// TwinCAT 3 PLC project MicroTestStandATM
// ProgramVersion: 3.1.4020.5
// libraries:
//   lcls-twincat-motion, * (SLAC)
//   lcls2-cc-lib, * (SLAC)
//   Tc2_Standard, * (Beckhoff Automation GmbH)
//   Tc2_System, * (Beckhoff Automation GmbH)
//   Tc2_Utilities, * (Beckhoff Automation GmbH)
//   Tc3_Module, * (Beckhoff Automation GmbH)
//   VisuDialogs
//   VisuSymbols,3.5.10.0,System
// project tree:
//   DUTs/ DUT_MotionStage_Extras.TcDUT (not stored)
//   / GlobalTextList.TcGTLO, PlcTask.TcTTO (not stored), VISU_TASK.TcTTO (not stored)
//   POUs/ Main.TcPOU
//   VISUs/ Visualization.TcVIS, VisualizationManager.TcVMO (not stored), VISU_MotionStage.TcVIS (not stored)
// real-time tasks:
//   TASK PlcTask: cycle T#1ms, priority 20, ADS port 350
//   TASK VISU_TASK: cycle T#200000us, priority 30, ADS port 351
// motion (NC):
//   TASK NC-Task 1 SAF: cycle T#1ms, priority 4, ADS port 501
//   TASK NC-Task 1 SVB: cycle T#1ms, priority 8, ADS port 511
//   AXIS MMS_Y (id 1)
//     Dynamic: AccelerationMaximum=200, DecelerationMaximum=200, Acceleration=200, Deceleration=200, Jerk=500, DelayTime=0.004
//     Velo: Maximum=65
//     TargetPosControl: Range=0.002, Time=0.25
//     OtherSettings: AllowMotionCmdToSlave=true
//     encoder EncType=29
//       EncPara: ScaleFactorNumerator=5e-05, Offset=-214686.941, MaxCount=#xffffffff, ReferenceSystem=1
//         Inc: RefSoftSyncMask=#x0000ffff
//     drive DrvType=24
//       Analog: VeloReferenz=100, ScaleFactorActTorque=0.1
//       TimeComp: TaskDelayCycles=1
//     controller CtrType=2
//       CtrPara: PriorControlFactor=1
//         PosDiffControl: Range=1
//         PID: PosKp=20, PosExtKp=1, PosExtVelo=0.1, DeadBandPosition=0.002
//         Observer: BandWidth=20
//   AXIS MMS_X (id 2)
//     Dynamic: AccelerationMaximum=200, DecelerationMaximum=200, Acceleration=200, Deceleration=200, Jerk=500
//     Velo: Maximum=10
//     OtherSettings: AllowMotionCmdToSlave=true
//     encoder EncType=29
//       EncPara: ScaleFactorNumerator=5e-05, MaxCount=#xffffffff, ReferenceSystem=1
//         Inc: RefSoftSyncMask=#x0000ffff
//     drive DrvType=24
//       Analog: VeloReferenz=15.875, ScaleFactorActTorque=0.1
//       TimeComp: TaskDelayCycles=1
//     controller CtrType=1
//       CtrPara: PriorControlFactor=1
//         PosDiffControl: Enable=false, Range=1
//         PID: PosKp=0
//         Observer: BandWidth=20
// I/O:
//   DEVICE Device 1 (EtherCAT)
// variable links:
//   (this object) <-> Device 1 (EtherCAT)/EK1100/EL5042
//     Enc/Inputs/In/nComState @bit 1 <-> WcState/InputToggle
//     Enc/Inputs/In/nComState <-> WcState/WcState
//     Enc/Inputs/In/nDataIn1 <-> FB Inputs Channel 1/Position
//     Enc/Inputs/In/nDataIn1 <-> FB Inputs Channel 2/Position
//     Enc/Inputs/In/nState1 @bit 12 <-> FB Inputs Channel 1/Status/Diag
//     Enc/Inputs/In/nState1 @bit 12 <-> FB Inputs Channel 2/Status/Diag
//     Enc/Inputs/In/nState1 @bit 1 <-> FB Inputs Channel 1/Status/Error
//     Enc/Inputs/In/nState1 @bit 1 <-> FB Inputs Channel 2/Status/Error
//     Enc/Inputs/In/nState1 @bit 14 <-> FB Inputs Channel 1/Status/Input cycle counter
//     Enc/Inputs/In/nState1 @bit 14 <-> FB Inputs Channel 2/Status/Input cycle counter
//     Enc/Inputs/In/nState1 @bit 2 <-> FB Inputs Channel 1/Status/Ready
//     Enc/Inputs/In/nState1 @bit 2 <-> FB Inputs Channel 2/Status/Ready
//     Enc/Inputs/In/nState1 @bit 13 <-> FB Inputs Channel 1/Status/TxPDO State
//     Enc/Inputs/In/nState1 @bit 13 <-> FB Inputs Channel 2/Status/TxPDO State
//     Enc/Inputs/In/nState1 <-> FB Inputs Channel 1/Status/Warning
//     Enc/Inputs/In/nState1 <-> FB Inputs Channel 2/Status/Warning
//   (this object) <-> Device 1 (EtherCAT)/EK1100/EL7041-Y
//     Drive/Inputs/In/nState1 @bit 3 <-> STM Status/Status/Error
//     Drive/Inputs/In/nState1 @bit 5 <-> STM Status/Status/Moving negative
//     Drive/Inputs/In/nState1 @bit 4 <-> STM Status/Status/Moving positive
//     Drive/Inputs/In/nState1 @bit 1 <-> STM Status/Status/Ready
//     Drive/Inputs/In/nState1 <-> STM Status/Status/Ready to enable
//     Drive/Inputs/In/nState1 @bit 6 <-> STM Status/Status/Torque reduced
//     Drive/Inputs/In/nState1 @bit 2 <-> STM Status/Status/Warning
//     Drive/Inputs/In/nState2 @bit 3 <-> STM Status/Status/Digital input 1
//     Drive/Inputs/In/nState2 @bit 4 <-> STM Status/Status/Digital input 2
//     Drive/Inputs/In/nState2 @bit 5 <-> STM Status/Status/Sync error
//     Drive/Inputs/In/nState2 @bit 7 <-> STM Status/Status/TxPDO Toggle
//     Drive/Inputs/In/nState4 @bit 1 <-> WcState/InputToggle
//     Drive/Inputs/In/nState4 <-> WcState/WcState
//     Drive/Outputs/Out/nCtrl1 <-> STM Control/Control/Enable
//     Drive/Outputs/Out/nCtrl1 @bit 2 <-> STM Control/Control/Reduce torque
//     Drive/Outputs/Out/nCtrl1 @bit 1 <-> STM Control/Control/Reset
//     Drive/Outputs/Out/nDataOut2[0] <-> STM Velocity/Velocity
//   (this object) <-> Device 1 (EtherCAT)/EK1100/EL7041-X
//     Drive/Inputs/In/nState1 @bit 3 <-> STM Status/Status/Error
//     Drive/Inputs/In/nState1 @bit 5 <-> STM Status/Status/Moving negative
//     Drive/Inputs/In/nState1 @bit 4 <-> STM Status/Status/Moving positive
//     Drive/Inputs/In/nState1 @bit 1 <-> STM Status/Status/Ready
//     Drive/Inputs/In/nState1 <-> STM Status/Status/Ready to enable
//     Drive/Inputs/In/nState1 @bit 6 <-> STM Status/Status/Torque reduced
//     Drive/Inputs/In/nState1 @bit 2 <-> STM Status/Status/Warning
//     Drive/Inputs/In/nState2 @bit 3 <-> STM Status/Status/Digital input 1
//     Drive/Inputs/In/nState2 @bit 4 <-> STM Status/Status/Digital input 2
//     Drive/Inputs/In/nState2 @bit 5 <-> STM Status/Status/Sync error
//     Drive/Inputs/In/nState2 @bit 7 <-> STM Status/Status/TxPDO Toggle
//     Drive/Inputs/In/nState4 @bit 1 <-> WcState/InputToggle
//     Drive/Inputs/In/nState4 <-> WcState/WcState
//     Drive/Outputs/Out/nCtrl1 <-> STM Control/Control/Enable
//     Drive/Outputs/Out/nCtrl1 @bit 2 <-> STM Control/Control/Reduce torque
//     Drive/Outputs/Out/nCtrl1 @bit 1 <-> STM Control/Control/Reset
//     Drive/Outputs/Out/nDataOut2[0] <-> STM Velocity/Velocity
//   MicroTestStandATM Instance <-> Device 1 (EtherCAT)/EK1100/EL2004
//     PlcTask Outputs/Main.M1.bBrakeRelease <-> Channel 1/Output
//   MicroTestStandATM Instance <-> Device 1 (EtherCAT)/EK1100/EL3314
//     PlcTask Inputs/Main.fbWFS.fbThermoCouple1.bError <-> TC Inputs Channel 1/Status/Error
//     PlcTask Inputs/Main.fbWFS.fbThermoCouple2.bError <-> TC Inputs Channel 2/Status/Error
//     PlcTask Inputs/Main.fbWFS.fbThermoCouple1.bOverrange <-> TC Inputs Channel 1/Status/Overrange
//     PlcTask Inputs/Main.fbWFS.fbThermoCouple2.bOverrange <-> TC Inputs Channel 2/Status/Overrange
//     PlcTask Inputs/Main.fbWFS.fbThermoCouple1.bUnderrange <-> TC Inputs Channel 1/Status/Underrange
//     PlcTask Inputs/Main.fbWFS.fbThermoCouple2.bUnderrange <-> TC Inputs Channel 2/Status/Underrange
//     PlcTask Inputs/Main.fbWFS.fbThermoCouple1.iRaw <-> TC Inputs Channel 1/Value
//     PlcTask Inputs/Main.fbWFS.fbThermoCouple2.iRaw <-> TC Inputs Channel 2/Value
//   MicroTestStandATM Instance <-> Device 1 (EtherCAT)/EK1100/EL5042
//     PlcTask Inputs/Main.iM1RawEncoder <-> FB Inputs Channel 1/Position
//     PlcTask Inputs/Main.iM2RawEncoder <-> FB Inputs Channel 2/Position
//   MicroTestStandATM Instance <-> Device 1 (EtherCAT)/EK1100/EL7041-Y
//     PlcTask Inputs/Main.M1.bLimitBackwardEnable <-> STM Status/Status/Digital input 2
//     PlcTask Inputs/Main.M1.bLimitForwardEnable <-> STM Status/Status/Digital input 1
//   MicroTestStandATM Instance <-> NC-Task 1 SAF/Axes/MMS_X
//     PlcTask Inputs/Main.M2.Axis.NcToPlc <-> Outputs/ToPlc
//     PlcTask Outputs/Main.M2.Axis.PlcToNc <-> Inputs/FromPlc
//   MicroTestStandATM Instance <-> NC-Task 1 SAF/Axes/MMS_Y
//     PlcTask Inputs/Main.M1.Axis.NcToPlc <-> Outputs/ToPlc
//     PlcTask Outputs/Main.M1.Axis.PlcToNc <-> Inputs/FromPlc

// ---- POUs/Main.TcPOU
PROGRAM Main
VAR
	{attribute 'TcLinkTo' := '.bLimitForwardEnable  := TIIB[EL7041-Y]^STM Status^Status^Digital input 1;
	                          .bLimitBackwardEnable := TIIB[EL7041-Y]^STM Status^Status^Digital input 2;
	                          .bBrakeRelease        := TIIB[EL2004]^Channel 1^Output'}
	M1: DUT_MotionStage;
	M1_Extras: DUT_MotionStage_Extras;
    
	M2: DUT_MotionStage;
	M2_Extras: DUT_MotionStage_Extras;
	
	{attribute 'TcLinkTo' := '.fbThermoCouple1.bError := TIIB[EL3314]^TC Inputs Channel 1^Status^Error;
							  .fbThermoCouple1.bUnderrange := TIIB[EL3314]^TC Inputs Channel 1^Status^Underrange;
							  .fbThermoCouple1.bOverrange := TIIB[EL3314]^TC Inputs Channel 1^Status^Overrange;
							  .fbThermoCouple1.iRaw := TIIB[EL3314]^TC Inputs Channel 1^Value;
							  .fbThermoCouple2.bError := TIIB[EL3314]^TC Inputs Channel 2^Status^Error;
							  .fbThermoCouple2.bUnderrange := TIIB[EL3314]^TC Inputs Channel 2^Status^Underrange;
							  .fbThermoCouple2.bOverrange := TIIB[EL3314]^TC Inputs Channel 2^Status^Overrange;
							  .fbThermoCouple2.iRaw := TIIB[EL3314]^TC Inputs Channel 2^Value'}
	fbWFS: FB_WFS;
	

    {attribute 'TcLinkTo' := 'TIIB[EL5042]^FB Inputs Channel 1^Position'}
	iM1RawEncoder AT %I*: ULINT;
	iM1AdjustedEncoder: UDINT;
    
    {attribute 'TcLinkTo' := 'TIIB[EL5042]^FB Inputs Channel 2^Position'}
    iM2RawEncoder AT %I*: ULINT;
    iM2AdjustedEncoder: UDINT;
    
	iMaxLINT: ULINT := 18446744073709551615;
	
	bStartup: BOOL := TRUE;
END_VAR

fbWFS(
    stYStage := M1,
    stZStage := M2);
iM1AdjustedEncoder := ULINT_TO_UDINT(iMaxLINT - iM1RawEncoder) + 1;
iM2AdjustedEncoder := ULINT_TO_UDINT(iM2RawEncoder);

M1_Extras.bVisuHighLim := NOT M1.bAllForwardEnable;
M1_Extras.bVisuLowLim := NOT M1.bAllBackwardEnable;
M2_Extras.bVisuHighLim := NOT M2.bAllForwardEnable;
M2_Extras.bVisuLowLim := NOT M2.bAllBackwardEnable;

IF bStartup THEN
	bStartup := FALSE;
	M1.fVelocity := 20;
	M1.fAcceleration := 10;
	M1.fDeceleration := 10;
	M2.fVelocity := 5;
	M2.fAcceleration := 10;
	M2.fDeceleration := 50;
END_IF

END_PROGRAM

// ---- GlobalTextList.TcGTLO
TEXTLIST GlobalTextList
  593 = '%f'
  964 = '%X'
  957 = '+'
  951 = '-'
  960 = '0 = Default Acceleration'
  962 = '0 = Default Deceleration'
  959 = 'Acceleration: %f'
  504 = 'Cam Power'
  955 = 'Clear'
  582 = 'Close Screen'
  949 = 'Control'
  684 = 'Controls'
  594 = 'Current Position'
  961 = 'Deceleration: %f'
  324 = 'Encoder'
  965 = 'Error Code'
  963 = 'Error:'
  953 = 'GO'
  954 = 'GO to set position'
  595 = 'High Limit Hit Indicator'
  768 = 'Illuminator: %f %'
  592 = 'Low Limit Hit Indicator'
  30 = 'Motion Stage'
  460 = 'Motor'
  596 = 'Moving:'
  311 = 'Parker Stage'
  109 = 'PM TC: %f C'
  658 = 'PM Temp: %f C'
  598 = 'Power Meter: %f V'
  921 = 'PPM'
  890 = 'Raw count: %d'
  7 = 'Raw count: %f'
  274 = 'Readbacks'
  950 = 'Set Position'
  470 = 'Settings'
  591 = 'Status'
  952 = 'Step Size'
  956 = 'STOP'
  917 = 'Temp 1: %f C'
  256 = 'Temp 2: %f C'
  865 = 'Thermocouple Readback'
  151 = 'Thermocouple Readbacks'
  958 = 'Velocity: %f'
  562 = 'X Motor'
  568 = 'Y Motor'
  316 = 'Yag Temp: %f C'
  824 = 'Z Motor'
END_TEXTLIST

// ---- VISUs/Visualization.TcVIS
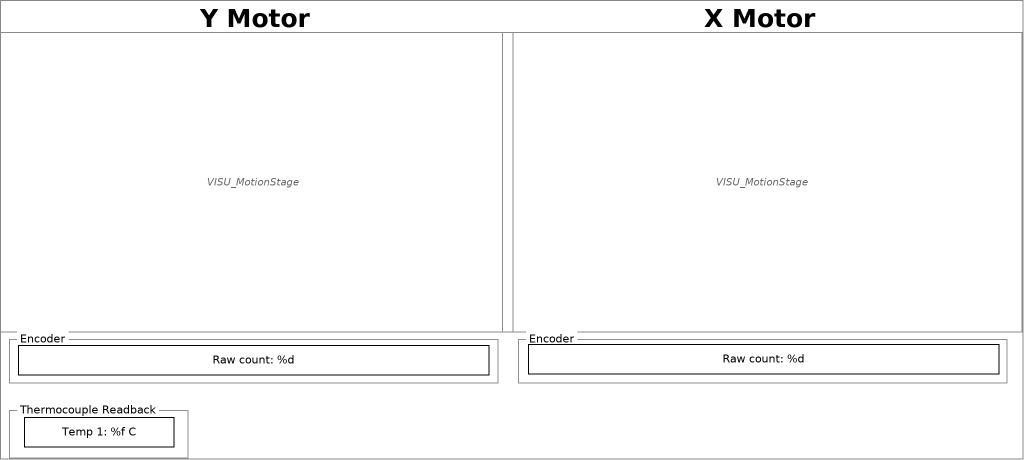
VISUALIZATION Visualization  // 1024x460
    Label (14,3 482x30), "Y Motor"
    Label (519,3 482x30), "X Motor"
    GroupBox (9,402 179x56), "Thermocouple Readback"
        Rectangle (15,15 150x30), "Temp 1: %f C", text variable: Main.fbWFS.fbThermoCouple1.fTemp
    Frame (-7,32 520x300)
        shows VISU_MotionStage(VisuMotionStage := Main.M1, Extras := Main.M1_Extras)
    Frame (502,32 520x300)
        shows VISU_MotionStage(VisuMotionStage := Main.M2, Extras := Main.M2_Extras)
    GroupBox (9,331 489x52), "Encoder"
        Rectangle (9,14 471x30), "Raw count: %d", text variable: Main.iM1AdjustedEncoder
    GroupBox (518,331 489x52), "Encoder"
        Rectangle (10,13 471x30), "Raw count: %d", text variable: Main.iM2AdjustedEncoder
END_VISUALIZATION
